// LS Electric XG5000 project: 동남119
// PLC NewPLC
// module base 0 slot 0: 입출력 모듈:XBC-DN/DP14E (DC 24V 입력 8점, 트랜지스터 출력 6점)

PROGRAM NewProgram (task: 스캔 프로그램)

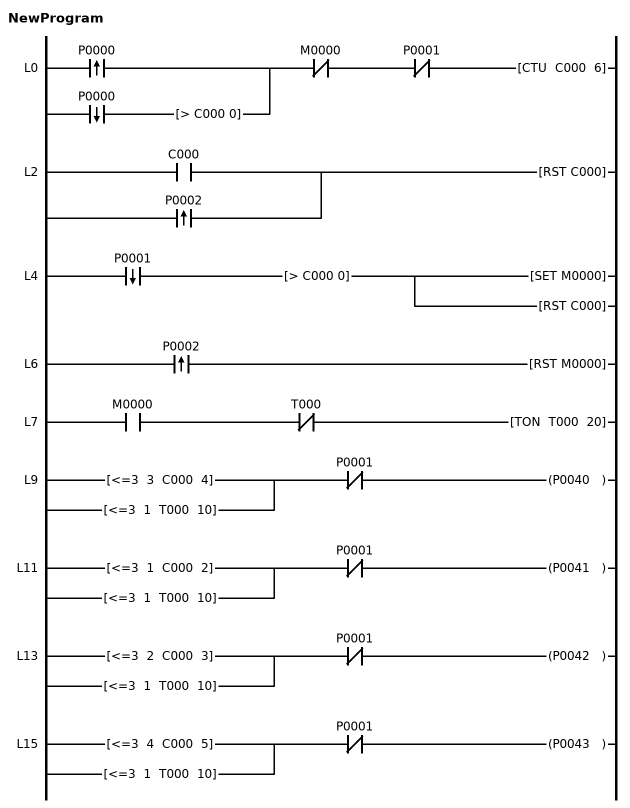
; L0
LOADP     P0000
LOADN     P0000
AND>      C000 0
OR LOAD
AND NOT   M0000
AND NOT   P0001
CTU       C000 6
; L2
LOAD      C000
ORP       P0002
RST       C000
; L4
LOADN     P0001
AND>      C000 0
SET       M0000
RST       C000
; L6
LOADP     P0002
RST       M0000
; L7
LOAD      M0000
AND NOT   T000
TON       T000 20
; L9
LOAD<=3   3 C000 4
OR<=3     1 T000 10
AND NOT   P0001
OUT       P0040
; L11
LOAD<=3   1 C000 2
OR<=3     1 T000 10
AND NOT   P0001
OUT       P0041
; L13
LOAD<=3   2 C000 3
OR<=3     1 T000 10
AND NOT   P0001
OUT       P0042
; L15
LOAD<=3   4 C000 5
OR<=3     1 T000 10
AND NOT   P0001
OUT       P0043